// Brief: Master Arm Orientation Matching
FUNCTION_BLOCK PUBLIC FB_ArmMatching EXTENDS FB_MasterArmCtrlBase
VAR_INPUT
END_VAR
VAR_OUTPUT
END_VAR
VAR
END_VAR

END_FUNCTION_BLOCK

(* stored: Version 1.1.0.1, ProductVersion 3.1.4024.12
   POU FB_ArmMatching: Id {886a3c3b-c6fb-4a12-8c63-bddb11202d66}, SpecialFunc None *)
